// TIA Portal V19 export
ORGANIZATION_BLOCK "Cyclic interrupt 100ms"   // OB30, LAD, CyclicInterrupt
{ S7_Optimized_Access := 'TRUE' }
// stored: SetENOAutomatically false
   VAR_INPUT
      Initial_Call : Bool;   // Initial call of this OB
      Event_Count : Int;   // Events discarded
   END_VAR
   VAR_TEMP
      i : Int;
   END_VAR
BEGIN
END_ORGANIZATION_BLOCK
